# EPICS substitutions: iocs/motorZynqIOC/motorZynqIOCApp/Db/motor.substitutions
file "$(MOTOR)/db/basic_asyn_motor.db"
{
pattern
{P,       N, M,             DTYP,        PORT,    ADDR, DESC,       EGU,  DHLM, DLLM, DIR, VMAX, VELO, VBAS, ACCL, BDST, BVEL, BACC, MRES,  RRES,  PREC, INIT}
{"$(Sys)",  1, "{$(Dev)-Ax:1}", "asynMotor", "$(Port)", 0,    "Motor 0",  rev,  0,    0,    Pos, 1.0,  0.5,  0.1,  0.5,  0,    1,    0.5,  0.005, 0.005, 3,    ""}
{"$(Sys)",  2, "{$(Dev)-Ax:2}", "asynMotor", "$(Port)", 1,    "Motor 1",  rev,  0,    0,    Pos, 1.0,  0.5,  0.1,  0.5,  0,    1,    0.5,  0.005, 0.005, 3,    ""}
{"$(Sys)",  3, "{$(Dev)-Ax:3}", "asynMotor", "$(Port)", 2,    "Motor 2",  rev,  0,    0,    Pos, 1.0,  0.5,  0.1,  0.5,  0,    1,    0.5,  0.005, 0.005, 3,    ""}
{"$(Sys)",  4, "{$(Dev)-Ax:4}", "asynMotor", "$(Port)", 3,    "Motor 3",  rev,  0,    0,    Pos, 1.0,  0.5,  0.1,  0.5,  0,    1,    0.5,  0.005, 0.005, 3,    ""}
}
